(* IEC 61131-3 sources: astools/Data/ASTemplates/Default/Export Dialog/LogicalView/Libraries/AsUSB, 3 files *)

(* ---- AsUSB.typ ---- *)
TYPE
    usbNode_typ			: STRUCT		(* statistics *)
	interfaceClass		: UINT;			(* Interface Class des USB Gerätes *)
	interfaceSubClass	: UINT;			(* Interface SubClass des USB Gerätes *)
	interfaceProtocol	: UINT;			(* Interface Protocol des USB Gerätes *)
	vendorId			: UINT;			(* Device Vendor ID *)
	productId			: UINT;			(* Device Product ID *)
	bcdDevice			: UINT;			(* USB device release version binary coded decimal *)
	ifName				: STRING[127];	(* USB IF Name *)
	END_STRUCT;
END_TYPE

TYPE
	usbDeviceDescr_typ	: STRUCT		(* statistics *)
    length				: USINT;		(* bLength *)
    descriptorType		: USINT;		(* bDescriptorType *)
    bcdUsb				: UINT;		    (* bcdUSB - USB release in BCD *)
    deviceClass			: USINT;	    (* bDeviceClass *)
    deviceSubClass		: USINT;		(* bDeviceSubClass *)
    deviceProtocol		: USINT;		(* bDeviceProtocol *)
    maxPacketSize0		: USINT;		(* bMaxPacketSize0 *)
    vendor				: UINT;			(* idVendor *)
    product				: UINT;			(* idProduct *)
    bcdDevice			: UINT;			(* bcdDevice - dev release in BCD *)
    manufacturerIndex	: USINT;		(* iManufacturer *)
    productIndex		: USINT;		(* iProduct *)
    serialNumberIndex	: USINT;		(* iSerialNumber *)
    numConfigurations	: USINT;		(* bNumConfigurations *)
	END_STRUCT;
END_TYPE

TYPE
	usbConfigDescr_typ	: STRUCT		(* statistics *)
	bLength				: USINT;		(* Size of this descriptor in bytes *)
    bDescriptorType		: USINT;		(* CONFIGURATION Descriptor Type *)
    wTotalLength		: UINT;			(* Configuration data length *)
    bNumInterfaces		: USINT;		(* Number of interfaces supported *)
    bConfigurationValue	: USINT;		(* SetConfiguration() function argument *)
    iConfiguration		: USINT;	   	(* Configuration string descriptor *)
    bmAttributes		: USINT;	    (* Bitmap configuration characteristics *)
    MaxPower			: USINT;		(* Max pwr consumption (mA) of operational device on bus *)
	END_STRUCT;
END_TYPE

TYPE
	usbStringDescr_typ	: STRUCT		(* statistics *)
    length				: USINT;		(* bLength *)
    descriptorType		: USINT;		(* bDescriptorType *)
    string				: STRING[1];	(* bString - variable len *)
	END_STRUCT;
END_TYPE

TYPE
	usbInterfaceDescr_typ	: STRUCT	(* statistics *)
    bLength					: USINT;	(* Size of this descriptor in bytes *)
    bDescriptorType			: USINT;	(* Interface Descriptor Type *)
    bInterfaceNumber		: USINT;	(* Zero-based interface number *)
    bAlternateSetting		: USINT;	(* Alternate setting for interface *)
    bNumEndpoints			: USINT;    (* Num of endpoints (excluding endpoint zero) *)
    bInterfaceClass			: USINT;	(* Class code of this interface *)
    bInterfaceSubClass		: USINT;	(* Subclass code of this interface *)
    bInterfaceProtocol		: USINT;	(* Interface protocol code *)
    iInterface				: USINT;	(* Interface string descriptor *)
	END_STRUCT;
END_TYPE

TYPE
	usbEndpointDescr_typ	: STRUCT	(* statistics *)
    bLength					: USINT;	(* Descriptor length in bytes *)
    bDescriptorType			: USINT;	(* Endpoint Descriptor type *)
    bEndpointAddress		: USINT;	(* Endpoint address on the USB device *)
    bmAttributes			: USINT;	(* Endpoint transfer, sych & usage types attr *)
    wMaxPacketSize			: UINT;		(* Endpoint max packet size *)
    bInterval				: USINT;	(* Polling interval for endpoint data xfer *)
	END_STRUCT;
END_TYPE

(* ---- AsUSB.fun ---- *)
{REDUND_CONTEXT} {REDUND_UNREPLICABLE} FUNCTION_BLOCK UsbNodeListGet			(* get USB node list *)
	VAR_INPUT
		enable			: BOOL;			(* fub enable *)
		pBuffer			: UDINT;		(* pointer to input buffer *)
		bufferSize		: UDINT;		(* max length of input buffer *)
		filterInterfaceClass : UINT;	(* filter for interface class *)
		filterInterfaceSubClass : UINT;	(* filter for interface subclass *)
	END_VAR
	VAR_OUTPUT
		status			: UINT;			(* status *)
		allNodes		: UDINT;		(* all usb nodes on target *)
		listNodes		: UDINT;		(* usb nodes in the list *)
		attachDetachCount:UDINT;		(* attach/deatch actions *)
	END_VAR
	VAR
        i_state			: UINT;			(* internal variable *)
		i_result		: UINT;			(* internal variable *)
        i_tmp			: UDINT;		(* internal variable *)
	END_VAR
END_FUNCTION_BLOCK
{REDUND_CONTEXT} {REDUND_UNREPLICABLE} FUNCTION_BLOCK UsbNodeGet 				(* get USB node description *)
	VAR_INPUT
		enable			: BOOL;			(* fub enable *)
		nodeId			: UDINT;		(* unique node identifier of USBNodeListGet *)
		pBuffer			: UDINT;		(* pointer to input buffer *)
		bufferSize		: UDINT;		(* max length of input buffer *)
	END_VAR
	VAR_OUTPUT
		status			: UINT;			(* status *)
	END_VAR
	VAR
        i_state			: UINT;			(* internal variable *)
		i_result		: UINT;			(* internal variable *)
        i_tmp			: UDINT;		(* internal variable *)
	END_VAR
END_FUNCTION_BLOCK
{REDUND_CONTEXT} {REDUND_UNREPLICABLE} FUNCTION_BLOCK UsbDescriptorGet			(* get USB node descriptor *)
	VAR_INPUT
		enable			: BOOL;			(* fub enable *)
		nodeId			: UDINT;		(* unique node identifier of USBNodeListGet *)
		requestType		: USINT;		(* reqeust type *)
		descriptorType	: USINT;		(* descriptor type *)
		descriptorIndex	: USINT;		(* descriptor index *)
		languageId		: UINT;			(* language unicode *)
		pBuffer			: UDINT;		(* pointer to input buffer *)
		bufferSize		: UINT;			(* max length of input buffer *)
	END_VAR
	VAR_OUTPUT
		status			: UINT;			(* status *)
		actSize			: UINT;			(* length of received data *)
	END_VAR
	VAR
        i_state			: UINT;			(* internal variable *)
		i_result		: UINT;			(* internal variable *)
        i_tmp			: UDINT;		(* internal variable *)
	END_VAR
END_FUNCTION_BLOCK
{REDUND_CONTEXT} {REDUND_UNREPLICABLE} FUNCTION_BLOCK UsbMsDeviceReady			(* get USB mass storage device ready status *)
	VAR_INPUT
		enable			: BOOL;			(* fub enable *)
		pIfName			: UDINT;		(* pointer to string of ifName of input buffer of USBNodeGet *)
	END_VAR
	VAR_OUTPUT
		status			: UINT;			(* status *)
		ready			: BOOL;			(* device ready status true/false *)
	END_VAR
	VAR
        i_state			: UINT;			(* internal variable *)
		i_result		: UINT;			(* internal variable *)
        i_tmp			: UDINT;		(* internal variable *)
	END_VAR
END_FUNCTION_BLOCK

(* ---- AsUSB.var ---- *)
VAR CONSTANT
	asusb_CLASS_CDC					: USINT	:= 2;  		(* USB Communications and CDC Control class code *)
	asusb_CLASS_HID					: USINT	:= 3;  		(* USB Human Interface Interfaces class code *)
	asusb_CLASS_PRINTER				: USINT	:= 7;		(* USB Printer class code *)
	asusb_CLASS_MASS_STORAGE		: USINT := 8;		(* USB Mass storage class code *)
	asusb_CLASS_HUB					: USINT := 9;		(* USB Hub class code *)
	asusb_CLASS_VENDOR_SPECIFIC		: USINT := 255;		(* USB Vendor specific *)

	asusb_SUBCLASS_PRINTER			: USINT := 1;		(* USB PRINTER subclass code *)
	asusb_SUBCLASS_HID_BOOT			: USINT := 1;		(* USB HID Boot *)
	asusb_SUBCLASS_UFI_COMMAND_SET	: USINT := 4;		(* USB UFI command set *)
	asusb_SUBCLASS_SCSI_COMMAND_SET : USINT := 6;		(* SCSI command set definition *)

	asusb_DEVICENAMELENGTH			: USINT := 128;

	asusb_USB_RT_DEVICE				: USINT := 0;		(* Requesttype for device *)
	asusb_USB_RT_INTERFACE			: USINT := 1;		(* Requesttype for interface *)
	asusb_USB_RT_ENDPOINT			: USINT := 2;		(* Requesttype for endpoint *)

	asusb_USB_RT_STANDARD			: USINT := 0;		(* Requesttype standard *)
	asusb_USB_RT_CLASS				: USINT := 32;		(* Requesttype class-specific *)
	asusb_USB_RT_VENDOR				: USINT := 64;		(* Requesttype vendor-specific *)

	asusb_USB_DESCR_DEVICE			: USINT := 1;		(* Specifies the DEVICE descriptor *)
	asusb_USB_DESCR_CONFIG			: USINT := 2;		(* Specifies the CONFIGURATION descriptor *)
	asusb_USB_DESCR_STRING			: USINT := 3;		(* Specifies a STRING descriptor *)
	asusb_USB_DESCR_INTERFACE		: USINT := 4;		(* Specifies an INTERFACE descriptor *)
	asusb_USB_DESCR_ENDPOINT		: USINT := 5;		(* Specifies an ENDPOINT  descriptor *)

	asusb_USB_UNICODE_ENGLISH		: UINT	:= 1033;	(* languageId unicode english *)

	asusbERR_USB_NOTFOUND			: UINT	:= 32900;   (* Es wurde kein USB Gerät gefunden keine USB Geräte angesteckt *)
	asusbERR_BUFSIZE				: UINT	:= 32901;	(* Die übergebene Speicherlänge ist zu klein Größeren Speicher reservieren  *)
	asusbERR_NULLPOINTER			: UINT	:= 32902;	(* pBuffer ist nicht gesetzt pBuffer setzen *)

END_VAR
